Fanuc KAREL source: KA00052.KL

PROGRAM KA00052
%NOLOCKGROUP
VAR
  SRC: POSITION
  DST: STRING[80]
BEGIN
  DST = SRC
END KA00052
